// TIA Portal V18 export
DATA_BLOCK "OP010_MES_RecipeDB"   // DB9
{ S7_Optimized_Access := 'FALSE' }
   VAR
      Download : Bool;
      Downloading : Bool;
      LastTypeID : Int;
      DownloadDone : Bool;
      ParameterElement : Struct
         TypeName : String[50] := '';   // System Defined=
         TypeID : USInt := 0;   // System define= product type for parameters of servo ,press and so on
         B1PressProgram : Int := 0;
         B2PressProgram : Int := 0;
         CGlueShaftIV3Program_1 : Word := 0;
         CGlueShaftIV3Program_2 : Word := 0;
         CGlueShaftIV3Program_3 : Word := 0;
         CGlueShaftIV3Program_4 : Word := 0;
         CGlueMagnetIV3Program : Word := 0;
         CGlueProgram : Int := 0;
      END_STRUCT;
   END_VAR
BEGIN
END_DATA_BLOCK
